// TIA Portal V19 export
FUNCTION "DOL Control" : Void   // FC8, LAD
{ S7_Optimized_Access := 'TRUE' }
// stored: SetENOAutomatically false
   VAR_TEMP   // added for the SCL form of the ladder/FBD networks
      _w1 : Bool;
   END_VAR
BEGIN

REGION Network 1: Request Cooling Motor Run
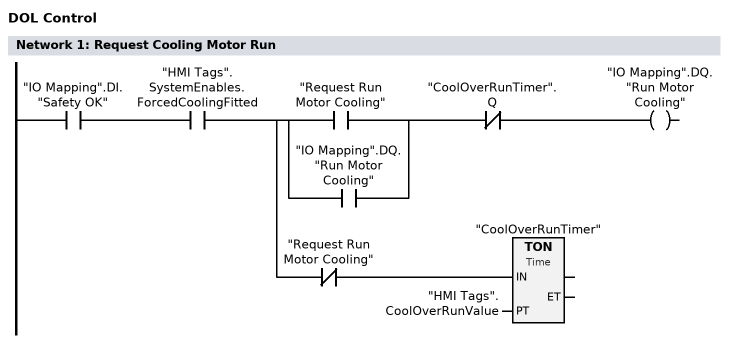
   RUNG wire#powerrail
      Contact( "IO Mapping".DI."Safety OK" )
      Contact( "HMI Tags".SystemEnables.ForcedCoolingFitted )
      wire#w1
      Contact( "Request Run Motor Cooling" )
      wire#w2
      I_Contact( "CoolOverRunTimer".Q )
      Coil( "IO Mapping".DQ."Run Motor Cooling" )
   END_RUNG
   RUNG wire#w1
      Contact( "IO Mapping".DQ."Run Motor Cooling" )
   END_RUNG wire#w2
   RUNG wire#w1
      I_Contact( "Request Run Motor Cooling" )
      { S7_Templates := "time_type := Time" } "CoolOverRunTimer".TON(pt := "HMI Tags".CoolOverRunValue, et =>)
   END_RUNG
   // the same network as SCL:
   #_w1 := "IO Mapping".DI."Safety OK" AND "HMI Tags".SystemEnables.ForcedCoolingFitted;
   "IO Mapping".DQ."Run Motor Cooling" := #_w1 AND ("Request Run Motor Cooling" OR "IO Mapping".DQ."Run Motor Cooling") AND NOT "CoolOverRunTimer".Q;
   "CoolOverRunTimer".TON(IN := #_w1 AND NOT "Request Run Motor Cooling", PT := "HMI Tags".CoolOverRunValue);
END_REGION
END_FUNCTION
